FUNCTION_BLOCK FB_WeighingStation IMPLEMENTS I_WorkingStation
VAR_INPUT
END_VAR
VAR_OUTPUT
END_VAR
VAR
END_VAR

{warning 'add property implementation'}
PROPERTY prTableRotationInterlock : BOOL
GET
END_GET
SET
END_SET
END_PROPERTY

{warning 'add property implementation'}
PROPERTY prTableRotationRequest : BOOL
GET
END_GET
SET
END_SET
END_PROPERTY

END_FUNCTION_BLOCK

(* stored: Version 1.1.0.1, ProductVersion 3.1.4024.15
   POU FB_WeighingStation: Id {44fe5b5a-0f0b-4511-b67e-0a0f72747565}, SpecialFunc None
   Property prTableRotationInterlock: Id {a3bd4f2e-7fc9-48a1-a0b6-851ef9873feb}
   Get Get: Id {43e5f169-a4d0-4c8e-91de-42b275f24a50}
   Set Set: Id {76b95d3b-5bcf-4249-9d73-08c145522c05}
   Property prTableRotationRequest: Id {9ba3f7f5-258e-4771-a282-88d0ed0f827d}
   Get Get: Id {6fac5f09-d7bd-4453-b0f2-ad728a049eaf}
   Set Set: Id {6f2e0132-c59b-475b-ac07-1e59a09efec3} *)
